// TIA Portal V16 export
// export: Created 2021-07-12T14:47:20.6604663Z, ExportSetting WithDefaults, DisplayName Totally Integrated Automation Portal, DisplayVersion V16, DisplayName TIA Portal Version Control Interface, DisplayVersion V16, DisplayName TIA Portal Openness, DisplayVersion V16, DisplayName STEP 7 Professional, DisplayVersion V16, DisplayName STEP 7 Safety, DisplayVersion V16, DisplayName WinCC Professional, DisplayVersion V16
TYPE "SimaHydTO_typeHMIConnectionAxisToDataAxisUnits"
TITLE = SimaHydTO_typeHMIConnectionAxisToDataAxisUnits
// HMI interface: Technology object axis units
// stored: IsFailsafeCompliant false
   STRUCT
      lengthUnit : UDInt := 0;
      velocityUnit : UDInt := 0;
      forceUnit : UDInt := 0;
      timeUnit : UDInt := 1054;
   END_STRUCT;
END_TYPE
